// TIA Portal V20 export
FUNCTION "Program_1" : Void   // FC1, LAD
{ S7_Optimized_Access := 'TRUE' }
// stored: SetENOAutomatically false
BEGIN

REGION Network 1
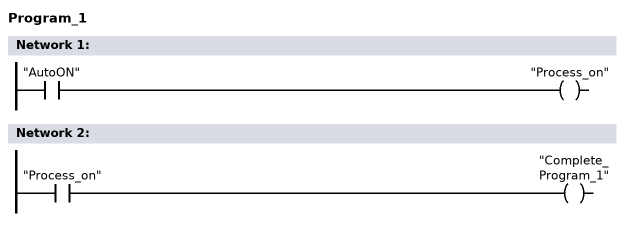
   RUNG wire#powerrail
      Contact( "AutoON" )
      Coil( "Process_on" )
   END_RUNG
   // the same network as SCL:
   "Process_on" := "AutoON";
END_REGION

REGION Network 2
   RUNG wire#powerrail
      Contact( "Process_on" )
      Coil( "Complete_Program_1" )
   END_RUNG
   // the same network as SCL:
   "Complete_Program_1" := "Process_on";
END_REGION
END_FUNCTION
